RoboDK station: PJT(test).rdk

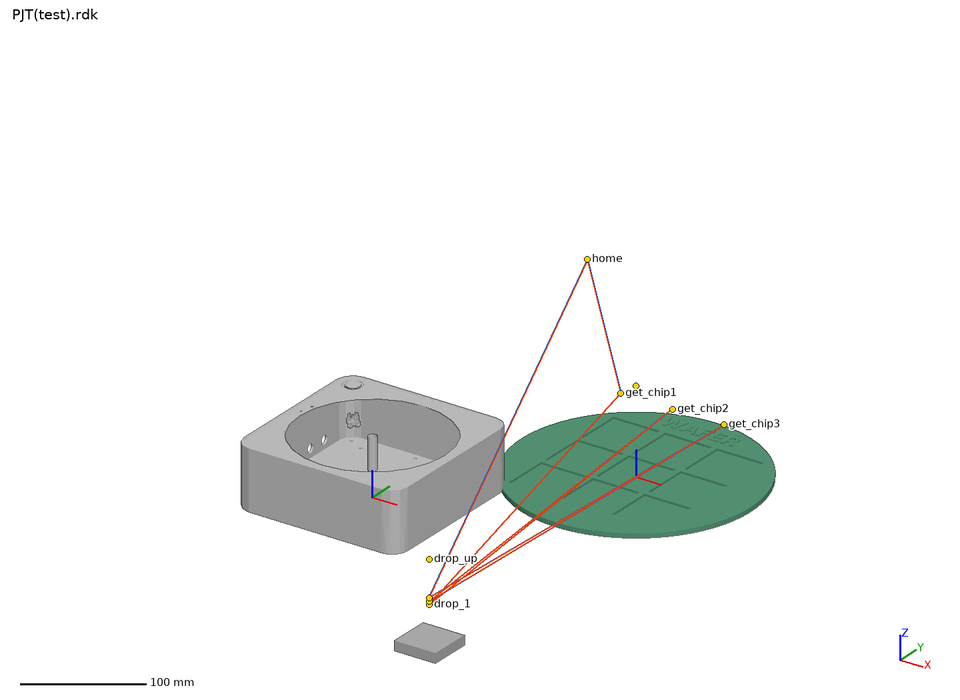
[picture v0: the station drawn from its stored meshes, robots at their saved joint values, targets as dots, program paths as lines]
Station PJT(test) (saved by RoboDK 5.8.0). Poses are relative to the parent item; angles as X-Y-Z fixed-axis rotations.
  - frame Dobot Magician Base at (0, 0, 0) mm
    - robot Dobot Magician: 4 axes, payload 0.5 kg, reach 320 mm, repeatability 0.2 mm, weight 4 kg
        joint limits [-90, -0.001, -10, -90] to [90, 85, 95, 90]; home [0, 0, 0, 0]; saved at [-87.048, 32.523, 55.51, 0]
      - tool Tool 1, TCP at (0, 0, 0) mm
  - frame WAFER at (150, 150, 0) mm
    - object chip_case3-3 at (0, 0, 0) mm, size 220 x 220 x 5 mm, geometry from chip_case3-3.stl
    - target get_chip3 (Cartesian target) at (50, 50, 40) mm, rotated rx 180 ry 0 rz -180 deg; joints [45, 79.759, 52.743, 45] of Dobot Magician
    - target get_chip2 (Cartesian target) at (0, 49.99, 39.99) mm, rotated rx 180 ry 0 rz 180 deg; joints [53.13, 72.31, 65.75, 53.13] of Dobot Magician
    - target get_chip1 (Cartesian target) at (-49.98, 50, 39.99) mm, rotated rx 180 ry 0 rz 180 deg; joints [63.43, 68.59, 75.45, 63.43] of Dobot Magician
    - target get_up (Cartesian target) at (0, 0, 80) mm, rotated rx 180 ry 0 rz -180 deg; joints [45, 50.317, 71.256, 45] of Dobot Magician
    - target drop_1 (Cartesian target) at (45, -350, 40) mm, rotated rx 180 ry 0 rz -180 deg; joints [-45.725, 78.774, 54.237, -45.725] of Dobot Magician
    - target drop_2 (Cartesian target) at (45, -350, 43) mm, rotated rx 180 ry 0 rz -180 deg; joints [-45.725, 77.644, 53.975, -45.725] of Dobot Magician
    - target drop_3 (Cartesian target) at (45, -350, 46) mm, rotated rx 180 ry 0 rz -180 deg; joints [-45.725, 76.525, 53.69, -45.725] of Dobot Magician
    - target drop_up (Cartesian target) at (45, -350, 80) mm, rotated rx 180 ry 0 rz -180 deg; joints [-45.725, 64.57, 49.016, -45.725] of Dobot Magician
    - target home (Cartesian target) at (58, -150, 268) mm, rotated rx 180 ry 0 rz -180 deg; joints [0, 0, 0, 0] of Dobot Magician
  - frame Frame 3 at (814.94, 1000, 0) mm
    - object root at (0, 0, 0) mm, size 200 x 200 x 50 mm, geometry from root.stl
    - object rota_1 at (0, 0, 20) mm, size 150 x 149.8 x 189.9 mm, geometry from rota_1.stl
    - object rota_21 at (30, 0, 150) mm, rotated rx 0 ry -90 rz 0 deg, size 50 x 295.8 x 40 mm, geometry from rota_2.stl
    - object rota_22 at (-10, 245, 150) mm, rotated rx 0 ry 90 rz 0 deg, size 50 x 295.8 x 40 mm, geometry from rota_2.stl
    - object rota_3 at (20, 490, 150) mm, rotated rx 0 ry 0 rz 90 deg, size 87.9 x 30 x 55 mm, geometry from rota_3.stl
  - Python program test (listed below)
  - program get-drop (15 instructions, listed below)
  - program re -get-drop (15 instructions, listed below)
  - object chip(4-4)(1) at (194.98, -200, 2.01) mm, size 40 x 40 x 3 mm, geometry from chip(4-4).stl
  - object chip(4-4)(2) at (195, -199.99, 5.01) mm, size 40 x 40 x 3 mm, geometry from chip(4-4).stl
  - object chip(4-4)(3) at (195, -200, 8) mm, size 40 x 40 x 3 mm, geometry from chip(4-4).stl
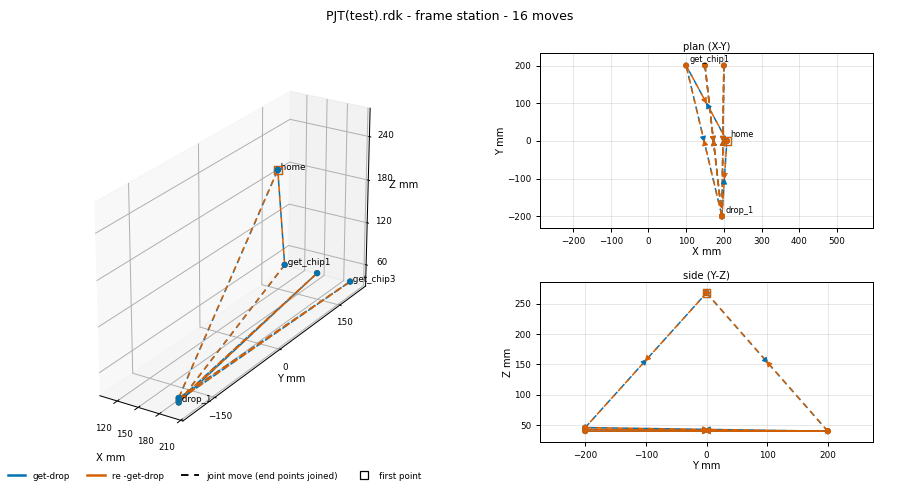
[picture p0: tool path of PJT(test).rdk in frame station, 16 of 16 moves have a stored position in this frame; points joined in program order, loops and branches not executed]

--- Python program test ---
from robodk import robolink    # RoboDK API
from robodk import robomath    # Robot toolbox
RDK = robolink.Robolink()

from robodk import *      # RoboDK API
from robolink import *    # Robot toolbox

import socket

# 연결된 RoboDK API 초기화
RDK = robolink.Robolink()

# 로봇과 관련된 Item 가져오기
RB1 = RDK.Item("Dobot Magician", itemtype=2)  # Dobot Magician 로봇

# 소켓 서버 설정
HOST = '0.0.0.0'  # 서버 IP 주소 (로봇이 실행되는 컴퓨터의 IP)
PORT = 10000            # 서버 포트 번호

# 조인트 범위 설정
JOINT_LIMITS = [
    (-90, 90),      # 1번 조인트
    (0.0, 85),      # 2번 조인트
    (-10, 95),      # 3번 조인트
    (-90, 90)       # 4번 조인트 (4번째 축 기본값 사용)
]

def parse_joint_values(data):
    """수신된 데이터를 파싱하여 조인트 값을 리스트로 반환"""
    try:
        return [float(x) for x in data.decode('utf-8').strip().split(',')]
    except ValueError:
        print("Invalid joint data received:", data)
        return None

def validate_joint_values(joint_values):
    """조인트 값이 허용 범위 내에 있는지 확인"""
    for i, value in enumerate(joint_values):
        joint_min, joint_max = JOINT_LIMITS[i]
        if not (joint_min <= value <= joint_max):
            print(f"Error: Joint {i+1} value {value} is out of range ({joint_min}, {joint_max}).")
            return False
    return True

def main():
    # 소켓 서버 초기화
    server_socket = socket.socket(socket.AF_INET, socket.SOCK_STREAM)
    server_socket.bind((HOST, PORT))
    server_socket.listen(1)
    print(f"Listening for connections on {HOST}:{PORT}...")

    connection, client_address = server_socket.accept()
    print(f"Connection established with {client_address}")

    try:
        while True:
            # 데이터 수신
            data = connection.recv(1024)
            if not data:
                break

            print(f"Received data: {data}")
            joint_values = parse_joint_values(data)

            if joint_values and len(joint_values) == 3:
                # 값 검증
                if validate_joint_values(joint_values):
                    # 로봇 조인트 값을 설정 (4축 중 앞 3축만 사용)
                    print(f"Moving robot to: {joint_values}")
                    RB1.MoveJ(joint_values + [0])  # 4번째 축은 기본값(0) 설정
                else:
                    print("Invalid joint values received. Ignoring this command.")
            else:
                print("Invalid joint data length. Expected 3 values.")

    except KeyboardInterrupt:
        print("Server interrupted by user.")
    finally:
        connection.close()
        server_socket.close()
        print("Server closed.")

if __name__ == "__main__":
    main()

--- program get-drop (robot Dobot Magician) ---
  Set Ref.: WAFER
  MoveJ (home)
  MoveJ (get_chip1)
  Attach to Tool 1
  MoveJ (drop_1)
  Detach from Tool 1
  MoveJ (get_chip2)
  Attach to Tool 1
  MoveJ (drop_2)
  Detach from Tool 1
  MoveJ (get_chip3)
  Attach to Tool 1
  MoveJ (drop_3)
  Detach from Tool 1
  MoveJ (home)

--- program re -get-drop (robot Dobot Magician) ---
  Set Ref.: WAFER
  MoveJ (home)
  MoveJ (drop_3)
  Attach to Tool 1
  MoveJ (get_chip3)
  Detach from Tool 1
  MoveJ (drop_2)
  Attach to Tool 1
  MoveJ (get_chip2)
  Detach from Tool 1
  MoveJ (drop_1)
  Attach to Tool 1
  MoveJ (get_chip1)
  Detach from Tool 1
  MoveJ (home)
